KUKA KRL program: wkz4_ok.src, wkz4_ok.dat

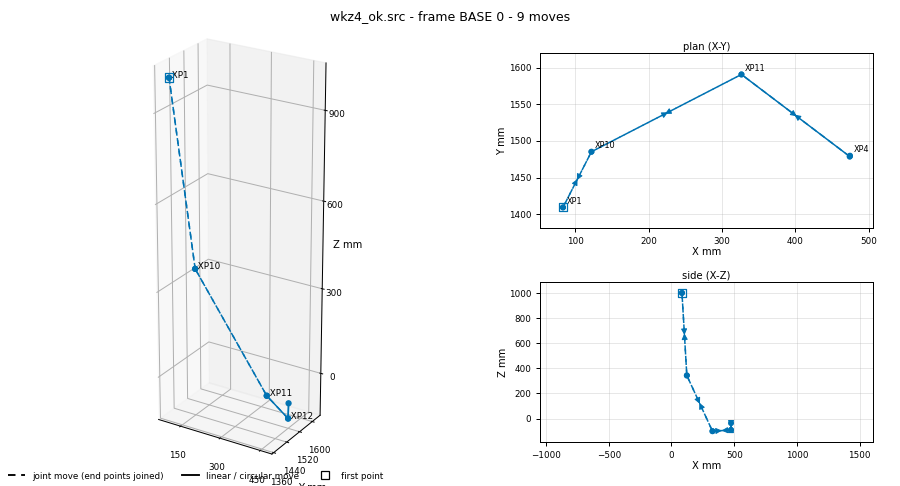
[picture p0: tool path of wkz4_ok.src in frame BASE 0, 9 of 9 moves have a stored position in this frame; points joined in program order, loops and branches not executed]
--- wkz4_ok.src ---
&ACCESS RVP
&REL 25
&COMMENT Check TCP C2
&PARAM TEMPLATE = C:\KRC\Roboter\Template\vorgabe
&PARAM EDITMASK = *
DEF wkz4_ok( )
;FOLD INI;%{PE}%V3.2.0,%MKUKATPBASIS,%CINIT,%VCOMMON,%P
;FOLD BAS INI;%{E}%V3.2.0,%MKUKATPBASIS,%CINIT,%VINIT,%P
GLOBAL INTERRUPT DECL 3 WHEN $STOPMESS==TRUE DO IR_STOPM ( )
INTERRUPT ON 3
BAS (#INITMOV,0 )
;ENDFOLD (BAS INI)
;FOLD A20 INI;%{E}%V3.2.0,%MKUKATPA20,%CINIT,%VINIT,%P
IF ARC20==TRUE THEN
A20 (ARC_INI)
INTERRUPT DECL 6 WHEN $CYCFLAG[3]==FALSE DO A20(TECH_STOP2)
ENDIF
;ENDFOLD (A20 INI)
;FOLD A10 INI;%{E}%V3.2.0,%MKUKATPARC,%CINIT,%VINIT,%P
IF A10_OPTION==#ACTIVE THEN
INTERRUPT DECL 4 WHEN $CYCFLAG[2]==FALSE DO A10 (#APPL_ERROR)
INTERRUPT DECL 7 WHEN A_ARC_SWI==#ACTIVE DO A10 (#ARC_SEAM)
INTERRUPT DECL 5 WHEN A_FLY_ARC==TRUE DO A10 (#HPU_ARC)
INTERRUPT  ON 5
A10_INI ( )
ENDIF
;ENDFOLD (A10 INI)
;FOLD GRIPPER INI;%{E}%V3.2.0,%MKUKATPGRIPPER,%CINIT,%VINIT,%P
USER_GRP(0,DUMMY,DUMMY,GDEFAULT)
;ENDFOLD (GRIPPER INI)
;FOLD SPOT INI;%{E}%V3.2.0,%MKUKATPSPOT,%CINIT,%VINIT,%P
USERSPOT(#INIT)
;ENDFOLD (SPOT INI)
;FOLD TOUCHSENSE INI;%{E}%V3.2.0,%MKUKATPTS,%CINIT,%VINIT,%P
IF H70_OPTION THEN
INTERRUPT DECL 15 WHEN $MEAS_PULSE[TOUCH_I[TOUCH_ACTIVE].IN_NR] DO H70 (6,CD0 )
INTERRUPT DECL 16 WHEN $ZERO_MOVE DO H70 (7,CD0 )
INTERRUPT DECL 17 WHEN $TECHPAR_C[FG_TOUCH,8]>0.5 DO H70 (8,CD0)
H70 (1,CD0 )
ENDIF
;ENDFOLD (TOUCHSENSE INI)
;FOLD USER INI;%{E}%V3.2.0,%MKUKATPUSER,%CINIT,%VINIT,%P
;Make your modifications here
;ENDFOLD (USER INI)
;ENDFOLD (INI)

; Caracterização dos meios de produção:
; Versão Atual:
; 14/09/2015 12:00 Name: P13.060-R3 CHANGES: Check TCP C2

chk_w4_wechs_ok ( )        ;VERIFICAÇÃO DE FERRAMENTA: c2

;FOLD PTP P1  Vel= 100 % PDAT1 Tool[4]:Gun C2 Base[0];%{PE}%R 4.1.16,%MKUKATPBASIS,%CMOVE,%VPTP,%P 1:PTP, 2:P1, 3:, 5:100, 7:PDAT1
$BWDSTART = FALSE
PDAT_ACT=PPDAT1
BAS(#PTP_DAT)
FDAT_ACT=FP1
BAS(#FRAMES)
BAS(#VEL_PTP,100)
PTP XP1
;ENDFOLD
;FOLD PTP P10 CONT Vel= 100 % PDAT10 Tool[4]:Gun C2 Base[0];%{PE}%R 4.1.16,%MKUKATPBASIS,%CMOVE,%VPTP,%P 1:PTP, 2:P10, 3:C_PTP, 5:100, 7:PDAT10
$BWDSTART = FALSE
PDAT_ACT=PPDAT10
BAS(#PTP_DAT)
FDAT_ACT=FP10
BAS(#FRAMES)
BAS(#VEL_PTP,100)
PTP XP10 C_PTP
;ENDFOLD
;FOLD PTP P11 CONT Vel= 100 % PDAT11 Tool[4]:Gun C2 Base[0];%{PE}%R 4.1.16,%MKUKATPBASIS,%CMOVE,%VPTP,%P 1:PTP, 2:P11, 3:C_PTP, 5:100, 7:PDAT11
$BWDSTART = FALSE
PDAT_ACT=PPDAT11
BAS(#PTP_DAT)
FDAT_ACT=FP11
BAS(#FRAMES)
BAS(#VEL_PTP,100)
PTP XP11 C_PTP
;ENDFOLD
;FOLD LIN P12  Vel= 1 m/s CPDAT3 Tool[4]:Gun C2 Base[0];%{PE}%R 4.1.16,%MKUKATPBASIS,%CMOVE,%VLIN,%P 1:LIN, 2:P12, 3:, 5:1, 7:CPDAT3
$BWDSTART = FALSE
LDAT_ACT=LCPDAT3
BAS(#CP_DAT)
FDAT_ACT=FP12
BAS(#FRAMES)
BAS(#VEL_CP,1)
LIN XP12
;ENDFOLD

;FOLD LIN P4  Vel= 1 m/s CPDAT2 Tool[4]:Gun C2 Base[0];%{PE}%R 4.1.16,%MKUKATPBASIS,%CMOVE,%VLIN,%P 1:LIN, 2:P4, 3:, 5:1, 7:CPDAT2
$BWDSTART = FALSE
LDAT_ACT=LCPDAT2
BAS(#CP_DAT)
FDAT_ACT=FP4
BAS(#FRAMES)
BAS(#VEL_CP,1)
LIN XP4
;ENDFOLD
;FOLD WAIT Time= 5 sec;%{PE}%R 4.1.16,%MKUKATPBASIS,%CWAIT,%VWAIT,%P 2:5
WAIT SEC 5
;ENDFOLD

;FOLD LIN P13  Vel= 1 m/s CPDAT4 Tool[4]:Gun C2 Base[0];%{PE}%R 4.1.16,%MKUKATPBASIS,%CMOVE,%VLIN,%P 1:LIN, 2:P13, 3:, 5:1, 7:CPDAT4
$BWDSTART = FALSE
LDAT_ACT=LCPDAT4
BAS(#CP_DAT)
FDAT_ACT=FP13
BAS(#FRAMES)
BAS(#VEL_CP,1)
LIN XP13
;ENDFOLD
;FOLD PTP P14 CONT Vel= 100 % PDAT12 Tool[4]:Gun C2 Base[0];%{PE}%R 4.1.16,%MKUKATPBASIS,%CMOVE,%VPTP,%P 1:PTP, 2:P14, 3:C_PTP, 5:100, 7:PDAT12
$BWDSTART = FALSE
PDAT_ACT=PPDAT12
BAS(#PTP_DAT)
FDAT_ACT=FP14
BAS(#FRAMES)
BAS(#VEL_PTP,100)
PTP XP14 C_PTP
;ENDFOLD
;FOLD PTP P15 CONT Vel= 100 % PDAT13 Tool[4]:Gun C2 Base[0];%{PE}%R 4.1.16,%MKUKATPBASIS,%CMOVE,%VPTP,%P 1:PTP, 2:P15, 3:C_PTP, 5:100, 7:PDAT13
$BWDSTART = FALSE
PDAT_ACT=PPDAT13
BAS(#PTP_DAT)
FDAT_ACT=FP15
BAS(#FRAMES)
BAS(#VEL_PTP,100)
PTP XP15 C_PTP
;ENDFOLD
;FOLD PTP P16  Vel= 100 % PDAT14 Tool[4]:Gun C2 Base[0];%{PE}%R 4.1.16,%MKUKATPBASIS,%CMOVE,%VPTP,%P 1:PTP, 2:P16, 3:, 5:100, 7:PDAT14
$BWDSTART = FALSE
PDAT_ACT=PPDAT14
BAS(#PTP_DAT)
FDAT_ACT=FP16
BAS(#FRAMES)
BAS(#VEL_PTP,100)
PTP XP16
;ENDFOLD
END

--- wkz4_ok.dat ---
&ACCESS RVP
&REL 25
&COMMENT Check TCP C2
&PARAM TEMPLATE = C:\KRC\Roboter\Template\vorgabe
&PARAM EDITMASK = *
DEFDAT  WKZ4_OK
;FOLD EXTERNAL DECLARATIONS;%{PE}%V3.2.0,%MKUKATPBASIS,%CEXT,%VCOMMON,%P
;FOLD BAS EXT;%{PE}%V3.2.0,%MKUKATPBASIS,%CEXT,%VEXT,%P
EXT  BAS (BAS_COMMAND  :IN,REAL  :IN )
DECL INT SUCCESS
;ENDFOLD
;FOLD A10 EXT;%{E}%V3.2.0,%MKUKATPARC,%CEXT,%VEXT,%P
EXT  A10 (A_CMD_T  :IN,A_STRT_T  :IN,A_WELD_T  :IN,A_END_T  :IN,INT  :IN )
;ENDFOLD
;FOLD A20 EXT;%{E}%V3.2.0,%MKUKATPA20,%CEXT,%VEXT,%P
EXT  A20 (INT  :IN,WELD_ST  :IN,WELD_FI  :IN,INT  :IN )
;ENDFOLD
;FOLD GRIPPER EXT;%{E}%V3.2.0,%MKUKATPGRIPPER,%CEXT,%VEXT,%P
EXT  H50 (INT  :IN,INT  :IN,INT  :IN,GRP_TYP  :IN )
;ENDFOLD
;FOLD SPOT EXT;%{E}%V3.2.0,%MKUKATPSPOT,%CEXT,%VEXT,%P
EXT  USERSPOT (S_COMMAND  :IN,SPOT_TYPE  :IN )
;ENDFOLD
;FOLD TOUCHSENSE EXT;%{E}%V3.2.0,%MKUKATPTS,%CEXT,%VEXT,%P
EXT  H70 (INT  :IN,SRCH_TYP_2  :OUT,E6POS  :IN,SRCH_TYP_3  :IN,SRCH_TYP_2  :IN,SRCH_TYP_2  :IN,SRCH_TYP_2  :IN,SRCH_TYP_2  :IN,SRCH_TYP_2  :IN,INT  :IN )
;ENDFOLD
;FOLD USER EXT;%{E}%V3.2.0,%MKUKATPUSER,%CEXT,%VEXT,%P
;Make here your modifications
;ENDFOLD
;ENDFOLD

DECL BASIS_SUGG_T LAST_BASIS={POINT1[] "P16                     ",POINT2[] "P16                     ",CP_PARAMS[] "CPDAT4                  ",PTP_PARAMS[] "PDAT14                  ",CONT[] "                        ",CP_VEL[] "1                       ",PTP_VEL[] "100                     "}
DECL E6POS XP1={x 83.4869537,y 1409.47302,z 1000.80402,a -139.854599,b 21.4527206,c -21.9509697,s 2,t 11,e1 0.0,e2 0.0,e3 0.0,e4 0.0,e5 0.0,e6 0.0}
DECL FDAT FP1={TOOL_NO 4,BASE_NO 0,IPO_FRAME #BASE}
DECL PDAT PPDAT1={VEL 100.0,ACC 100.0,APO_DIST 100.0}
DECL E6POS XP2={x 956.321777,y 2092.05103,z -52.729641,a 0.149778098,b -2.49974108,c 2.50239301,s 2,t 3,e1 0.0,e2 0.0,e3 0.0,e4 0.0,e5 0.0,e6 0.0}
DECL FDAT FP2={TOOL_NO 1,BASE_NO 0,IPO_FRAME #BASE}
DECL PDAT PPDAT2={VEL 100.0,ACC 100.0,APO_DIST 10.0}
DECL E6POS XP3={x 440.717407,y 2292.90405,z -68.8219528,a 4.03611517,b 0.155776694,c -0.43122521,s 2,t 11,e1 0.0,e2 0.0,e3 0.0,e4 0.0,e5 0.0,e6 0.0}
DECL FDAT FP3={TOOL_NO 1,BASE_NO 0,IPO_FRAME #BASE}
DECL PDAT PPDAT3={VEL 100.0,ACC 100.0,APO_DIST 10.0}
DECL E6POS XP4={x 474.399597,y 1479.96106,z -36.6517487,a -132.8526,b 0.799901187,c -0.135289803,s 2,t 3,e1 0.0,e2 0.0,e3 0.0,e4 0.0,e5 0.0,e6 0.0}
DECL FDAT FP4={TOOL_NO 4,BASE_NO 0,IPO_FRAME #BASE}
DECL PDAT PPDAT4={VEL 100.0,ACC 100.0,APO_DIST 10.0}
DECL E6POS XP5={x 1029.36902,y 2090.97412,z -58.8508987,a 0.0900030434,b -2.62809706,c -0.138254195,s 2,t 3,e1 0.0,e2 0.0,e3 0.0,e4 0.0,e5 0.0,e6 0.0}
DECL FDAT FP5={TOOL_NO 1,BASE_NO 0,IPO_FRAME #BASE}
DECL PDAT PPDAT5={VEL 100.0,ACC 100.0,APO_DIST 10.0}
DECL E6POS XP6={x 458.801208,y 1574.98096,z 322.150391,a 63.2156792,b -8.08211517,c 1.89149106,s 2,t 11,e1 0.0,e2 0.0,e3 0.0,e4 0.0,e5 0.0,e6 0.0}
DECL FDAT FP6={TOOL_NO 1,BASE_NO 0,IPO_FRAME #BASE}
DECL PDAT PPDAT6={VEL 100.0,ACC 100.0,APO_DIST 10.0}
DECL E6POS XP7={x 458.759491,y 1694.45605,z 322.132202,a 63.2113113,b -8.07844925,c 1.88991499,s 2,t 11,e1 0.0,e2 0.0,e3 0.0,e4 0.0,e5 0.0,e6 0.0}
DECL FDAT FP7={TOOL_NO 1,BASE_NO 0,IPO_FRAME #BASE}
DECL PDAT PPDAT7={VEL 100.0,ACC 100.0,APO_DIST 10.0}
DECL LDAT LCPDAT2={VEL 2.0,ACC 90.0,APO_DIST 100.0,APO_FAC 50.0}
DECL E6POS XP8={x 1029.36902,y 2090.97412,z -58.8508987,a 0.0900030434,b -2.62809706,c -0.138254195,s 2,t 3,e1 0.0,e2 0.0,e3 0.0,e4 0.0,e5 0.0,e6 0.0}
DECL FDAT FP8={TOOL_NO 1,BASE_NO 0,IPO_FRAME #BASE}
DECL LDAT LCPDAT1={VEL 2.0,ACC 90.0,APO_DIST 100.0,APO_FAC 50.0}
DECL PDAT PPDAT8={VEL 100.0,ACC 80.0,APO_DIST 10.0}
DECL E6POS XP9={x 956.322998,y 2092.05298,z -52.7274094,a 0.149773493,b -2.49978495,c 2.50250006,s 2,t 3,e1 0.0,e2 0.0,e3 0.0,e4 0.0,e5 0.0,e6 0.0}
DECL FDAT FP9={TOOL_NO 1,BASE_NO 0,IPO_FRAME #BASE}
DECL PDAT PPDAT9={VEL 100.0,ACC 100.0,APO_DIST 10.0}
DECL E6POS XP10={x 122.254898,y 1485.29004,z 343.362701,a -136.181595,b 0.787189424,c -0.687230706,s 2,t 3,e1 0.0,e2 0.0,e3 0.0,e4 0.0,e5 0.0,e6 0.0}
DECL FDAT FP10={TOOL_NO 4,BASE_NO 0,IPO_FRAME #BASE}
DECL PDAT PPDAT10={VEL 100.0,ACC 100.0,APO_DIST 100.0}
DECL E6POS XP11={x 326.527496,y 1590.53796,z -100.718498,a -132.8508,b 0.801788688,c -0.1355616,s 2,t 3,e1 0.0,e2 0.0,e3 0.0,e4 0.0,e5 0.0,e6 0.0}
DECL FDAT FP11={TOOL_NO 4,BASE_NO 0,IPO_FRAME #BASE}
DECL PDAT PPDAT11={VEL 100.0,ACC 100.0,APO_DIST 10.0}
DECL E6POS XP12={x 473.986786,y 1478.80798,z -90.8919067,a -132.852005,b 0.800183773,c -0.135114595,s 2,t 3,e1 0.0,e2 0.0,e3 0.0,e4 0.0,e5 0.0,e6 0.0}
DECL FDAT FP12={TOOL_NO 4,BASE_NO 0,IPO_FRAME #BASE}
DECL LDAT LCPDAT3={VEL 2.0,ACC 90.0,APO_DIST 100.0,APO_FAC 50.0}
DECL E6POS XP13={x 473.986786,y 1478.80798,z -90.8919067,a -132.852005,b 0.800183773,c -0.135114595,s 2,t 3,e1 0.0,e2 0.0,e3 0.0,e4 0.0,e5 0.0,e6 0.0}
DECL FDAT FP13={TOOL_NO 4,BASE_NO 0,IPO_FRAME #BASE}
DECL LDAT LCPDAT4={VEL 2.0,ACC 90.0,APO_DIST 100.0,APO_FAC 50.0}
DECL E6POS XP14={x 326.549988,y 1590.54199,z -100.724297,a -132.854599,b 0.801906586,c -0.134669006,s 2,t 3,e1 0.0,e2 0.0,e3 0.0,e4 0.0,e5 0.0,e6 0.0}
DECL FDAT FP14={TOOL_NO 4,BASE_NO 0,IPO_FRAME #BASE}
DECL PDAT PPDAT12={VEL 100.0,ACC 100.0,APO_DIST 10.0}
DECL E6POS XP15={x 122.252098,y 1485.29199,z 343.36441,a -136.181793,b 0.787147701,c -0.687201917,s 2,t 3,e1 0.0,e2 0.0,e3 0.0,e4 0.0,e5 0.0,e6 0.0}
DECL FDAT FP15={TOOL_NO 4,BASE_NO 0,IPO_FRAME #BASE}
DECL PDAT PPDAT13={VEL 100.0,ACC 100.0,APO_DIST 10.0}
DECL E6POS XP16={x 83.4794235,y 1409.45898,z 1000.755,a -139.853897,b 21.4511795,c -21.9497204,s 2,t 11,e1 0.0,e2 0.0,e3 0.0,e4 0.0,e5 0.0,e6 0.0}
DECL FDAT FP16={TOOL_NO 4,BASE_NO 0,IPO_FRAME #BASE}
DECL PDAT PPDAT14={VEL 100.0,ACC 100.0,APO_DIST 10.0}
ENDDAT
